(* CoDeSys 2.3 export: FTURNOFFK16PUMP.EXP *)

(* POU K16/fTurnOffK16Pump, ST *)
FUNCTION fTurnOffK16Pump : BOOL
VAR_INPUT
	PumpID : USINT;
END_VAR
VAR
END_VAR
	fSetK16Pump(FALSE, PumpID);
END_FUNCTION
